FUNCTION_BLOCK CachedEntity IMPLEMENTS I_Entity, I_Debug;
VAR
	_nIdx		: UDINT;
	_iRegister	: I_CompRegister;
END_VAR

//FB_Init is always available implicitly and it is used primarily for initialization.
//The return value is not evaluated. For a specific influence, you can also declare the
//methods explicitly and provide additional code there with the standard initialization
//code. You can evaluate the return value.
METHOD FB_Init: BOOL
VAR_INPUT
    bInitRetains: BOOL; // TRUE: the retain variables are initialized (reset warm / reset cold)
    bInCopyCode: BOOL;  // TRUE: the instance will be copied to the copy code afterward (online change)
	
	iRegister	: I_CompRegister;
	refCache	: REFERENCE TO UDINT;
END_VAR
VAR
	_eResult	: Result;
END_VAR
IF iRegister = 0 THEN
	DebugMsg(THIS^, 'iRegister = 0!');
	RETURN;
END_IF

_iRegister := iRegister;

CASE _eResult := _RegisterEntity(THIS^, nIndex => _nIdx) OF 
	Ok:
		IF __ISVALIDREF(refCache) THEN
			IF refCache = 0 THEN
				refCache := _nIdx;
			ELSE
				DebugMsg(THIS^, 'refCache is already assigned!');
			END_IF
		ELSE
			DebugMsg(THIS^, 'refCache is invalid!');
		END_IF
	ELSE
		DebugMsg(THIS^, Tc2_Standard.CONCAT('_RegisterEntity(THIS^) failed with code: ', TO_STRING(_eResult)));
END_CASE
END_METHOD

METHOD Get : Result
VAR_INPUT
	nIndex		: UDINT;
END_VAR
VAR_OUTPUT
	iComp		: I_Component;
END_VAR
Get := _iRegister.Get(nIndex, iComp => iComp);
END_METHOD

PROPERTY Index : UDINT
GET
Index := _nIdx;
END_GET
END_PROPERTY

PROPERTY RegCap : UDINT
GET
RegCap := _iRegister.Cap;
END_GET
END_PROPERTY

PROPERTY RegLen : UDINT
GET
RegLen := _iRegister.Length;
END_GET
END_PROPERTY

END_FUNCTION_BLOCK

(* stored: Version 1.1.0.1
   POU CachedEntity: Id {a3bc54a9-d8d0-4248-bd3c-08cec694f9da}, SpecialFunc None
   Method Fb_init: Id {8539f55c-e2a7-4dfd-8610-02959cbdb372}
   Method Get: Id {91193c45-6ad6-4c71-9d3b-ca7f00f174dc}
   Property Index: Id {febb387a-3cf5-49c1-b5ae-b17c660fbe32}
   Get Get: Id {32584628-3b6d-434a-90f6-aa18cc94cab2}
   Property RegCap: Id {6270dd8d-2423-4b84-95fe-3ad4b86a2fa8}
   Get Get: Id {d7581ebe-1030-494f-b66b-2afa260c2bc0}
   Property RegLen: Id {07a1d259-605d-447d-9cf8-ce3f2baa3f39}
   Get Get: Id {661aea84-0a5d-4926-82e8-14c9c14b3e00} *)
